FUNCTION_BLOCK RegisterSkill (* Composite Function Block Type *)
  (* Standard: 61499-2 *)
  (* Version 0.0, 2/13/2024, midxav, template *)
  PACKAGE Main;
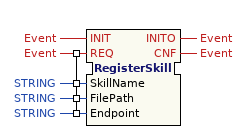
  EVENT_INPUT
    INIT;
    REQ WITH SkillName, FilePath, Endpoint;
  END_EVENT
  EVENT_OUTPUT
    INITO;
    CNF;
  END_EVENT
  VAR_INPUT
    SkillName : STRING;
    FilePath : STRING;
    Endpoint : STRING;
  END_VAR
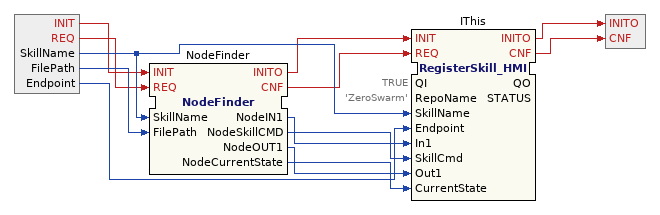
  FBS
    NodeFinder : NodeFinder;
    IThis : RegisterSkill_HMI(RepoName := 'ZeroSwarm', QI := TRUE);
  END_FBS
  EVENT_CONNECTIONS
    NodeFinder.INITO TO IThis.INIT;
    NodeFinder.CNF TO IThis.REQ;
    INIT TO NodeFinder.INIT;
    REQ TO NodeFinder.REQ;
    IThis.INITO TO INITO;
    IThis.CNF TO CNF;
  END_CONNECTIONS
  DATA_CONNECTIONS
    SkillName TO NodeFinder.SkillName;
    SkillName TO IThis.SkillName;
    NodeFinder.NodeIN1 TO IThis.In1;
    NodeFinder.NodeSkillCMD TO IThis.SkillCmd;
    NodeFinder.NodeOUT1 TO IThis.Out1;
    NodeFinder.NodeCurrentState TO IThis.CurrentState;
    FilePath TO NodeFinder.FilePath;
    Endpoint TO IThis.Endpoint;
  END_CONNECTIONS
END_FUNCTION_BLOCK
